// TIA Portal V20 export
DATA_BLOCK "instFB_AutoCtrl_Palletizing"   // DB
TITLE = instFB_AutoCtrl_Palletizing (C69 Phase 2.2)
VERSION : 1.1
// C69 Phase 2.2 (2026-05-18) — instance DB for FB_AutoCtrl_Palletizing. 48-element pts[] holds 16 boxes x 3 phases (approach/place/retract) for the 4-layer stacking pattern. instMoveLinAbs has NO AttributeList so SetPoint defaults to FALSE (required for MC_MoveLinearAbsolute Execute pulse to reach MC subsystem; lesson from Phase G C67 rev 0.1 failure).
// stored: InstanceOfName FB_AutoCtrl_Palletizing, InstanceOfType FB
"FB_AutoCtrl_Palletizing"
   // VAR
   //    sRTRIGInitialPath { S7_SetPoint := 'True'} : R_TRIG;
   //    sRTRIGStart { S7_SetPoint := 'True'} : R_TRIG;
   //    sRTRIGStop { S7_SetPoint := 'True'} : R_TRIG;
   //    instMoveLinAbs : MC_MOVELINEARABSOLUTE;
   //    pts { S7_SetPoint := 'True'} : Array[1..48] of "UDT_typePoint5";
   //    statTargetPos : "UDT_typePoint5";
   //    statOldStep : Int;
   //    statExecutePulse : Bool;
   //    statMoveDoneOld : Bool;
   //    statTotalDistance : LReal;
   //    statProgress : LReal;
   //    statActiveBoxes : Int;
   // END_VAR
BEGIN
END_DATA_BLOCK
